// TIA Portal V20 export
FUNCTION_BLOCK "FB_DigitalInput"   // FB15, SCL
{ S7_Optimized_Access := 'TRUE' }
// stored: AutoNumber false, MemoryReserve 100, SetENOAutomatically false
   VAR_INPUT
      iHWStatus { ExternalAccessible := 'False'; ExternalVisible := 'False'; ExternalWritable := 'False'} : Bool;   // PLC Digital Input Hardware status
   END_VAR
   VAR
      sDBI_F_Trig { S7_SetPoint := 'True'} : F_TRIG;
      sDBI_R_Trig { S7_SetPoint := 'True'} : R_TRIG;
      sSWStatus { ExternalAccessible := 'False'; ExternalVisible := 'False'; ExternalWritable := 'False'} : Bool;
      sSWPositiveFront { ExternalAccessible := 'False'; ExternalVisible := 'False'; ExternalWritable := 'False'} : Bool;
      sSWNegativeFront { ExternalAccessible := 'False'; ExternalVisible := 'False'; ExternalWritable := 'False'} : Bool;
   END_VAR
BEGIN
   REGION Description header 
       //==================================================================================
       // POSALUX Swiss SA / (C) Copyright 2024
       //----------------------------------------------------------------------------------
       // Title: Fonction Digital Input
       // Comment/Function: This function handles the state of a digital input, including
       //                   edge detection. It reads the hardware state, updates the
       //                   software state, and detects rising and falling edges.
       // Author: Gowsigan SRITHARAN
       // Engineering: TIA Portal v17
       //----------------------------------------------------------------------------------
       // Change log table:
       // Version  | Date     | Expert in charge | Changes applied
       // ---------|----------|------------------|-----------------------------------------
       // 00.00.01 | 20250106 | GSR              | First released version
       // =================================================================================
   END_REGION

   REGION Mise à jour de l'état de l'entree
       #sSWStatus:= #iHWStatus;
   END_REGION

   REGION Détection des fronts
       #sDBI_R_Trig(CLK := #sSWStatus,
                   Q => #sSWPositiveFront);

       #sDBI_F_Trig(CLK:=#sSWStatus,
                   Q=>#sSWNegativeFront);
   END_REGION
END_FUNCTION_BLOCK
